Yaskawa INFORM job: BATMAN_NEW2.JBI

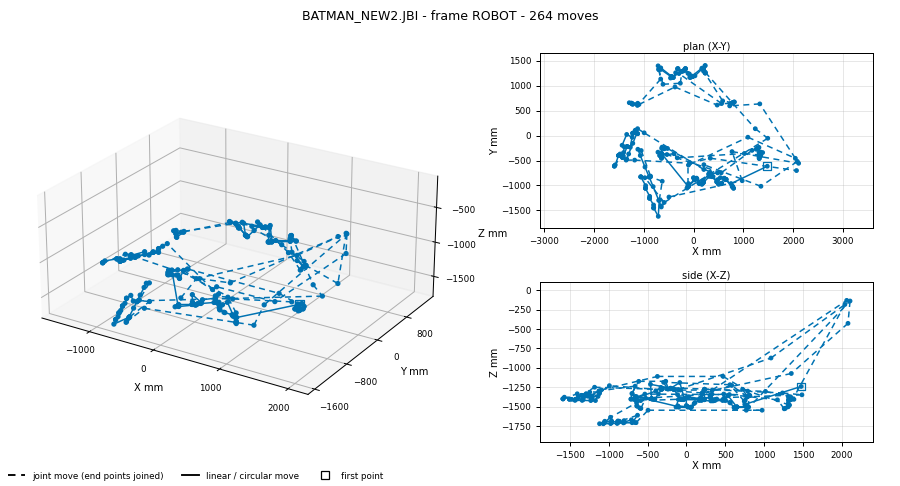
[picture p0: tool path of BATMAN_NEW2.JBI in frame ROBOT, 264 of 264 moves have a stored position in this frame; points joined in program order, loops and branches not executed]
/JOB
//NAME BATMAN_NEW2
///FOLDERNAME KRIS-SCIANA
//POS
///NPOS 316,316,264,16,0,0
///TOOL 0
///POSTYPE ROBOT
///RECTAN
///RCONF 0,0,0,0,0,0,0,0,0,0,0,0,0,0,0,0,0,0,0,0,0,0,0,0
C00000=1479.209,-614.254,-1239.827,11.6326,33.9671,-178.8219
C00001=751.878,-962.551,-1470.637,-9.9278,21.9341,47.3593
C00002=782.343,-1021.883,-1501.453,-6.5198,31.4589,38.6711
C00003=782.349,-1021.901,-1508.593,-6.5211,31.4595,38.6707
C00004=782.343,-1021.883,-1501.453,-6.5198,31.4589,38.6711
C00005=772.436,-1031.632,-1503.007,-6.5210,31.4603,38.6751
C00006=782.343,-1021.883,-1501.453,-6.5198,31.4589,38.6711
C00007=651.465,-878.509,-1502.529,-6.5193,31.4567,38.6726
C00008=649.681,-879.962,-1505.034,-6.5204,31.4570,38.6688
C00009=649.679,-879.971,-1512.967,-6.5216,31.4579,38.6721
C00010=649.681,-879.962,-1505.034,-6.5204,31.4570,38.6688
C00011=638.496,-885.487,-1507.904,-6.5213,31.4572,38.6690
C00012=649.681,-879.962,-1505.034,-6.5204,31.4570,38.6688
C00013=536.093,-844.110,-1358.224,-6.5194,31.4565,38.6698
C00014=485.208,-882.506,-1390.226,-6.5180,31.4566,38.6722
C00015=469.831,-925.588,-1412.310,-6.5196,31.4595,38.6720
C00016=469.838,-925.615,-1422.209,-6.5208,31.4607,38.6737
C00017=469.831,-925.588,-1412.310,-6.5196,31.4595,38.6720
C00018=460.916,-939.180,-1415.903,-6.5217,31.4610,38.6723
C00019=469.831,-925.588,-1412.310,-6.5196,31.4595,38.6720
C00020=390.944,-821.413,-1401.907,-6.5189,31.4593,38.6711
C00021=370.304,-823.702,-1415.949,-6.5184,31.4594,38.6679
C00022=370.309,-823.695,-1427.366,-6.5174,31.4589,38.6696
C00023=370.304,-823.702,-1415.949,-6.5184,31.4594,38.6679
C00024=362.481,-832.843,-1419.419,-6.5181,31.4591,38.6684
C00025=370.304,-823.702,-1415.949,-6.5184,31.4594,38.6679
C00026=304.377,-775.536,-1384.314,-6.5183,31.4594,38.6652
C00027=190.919,-901.974,-1384.308,6.6118,30.8401,128.8238
C00028=195.878,-934.762,-1411.685,6.6092,30.8405,128.8212
C00029=195.887,-934.767,-1420.325,6.6101,30.8407,128.8263
C00030=195.878,-934.762,-1411.685,6.6092,30.8405,128.8212
C00031=202.495,-948.084,-1414.851,6.6099,30.8403,128.8223
C00032=195.878,-934.762,-1411.685,6.6092,30.8405,128.8212
C00033=-1.386,-846.899,-1381.133,6.6069,30.8405,134.1399
C00034=-1.384,-846.902,-1485.292,6.6071,30.8406,134.1408
C00035=18.120,-884.199,-1503.049,6.6086,30.8410,134.1399
C00036=18.115,-884.194,-1511.506,6.6087,30.8409,134.1387
C00037=18.120,-884.199,-1503.049,6.6086,30.8410,134.1399
C00038=26.172,-895.008,-1505.663,6.6092,30.8415,134.1385
C00039=18.120,-884.199,-1503.049,6.6086,30.8410,134.1399
C00040=-111.813,-1001.782,-1489.786,6.6089,30.8396,134.1409
C00041=-110.516,-1020.985,-1499.218,6.6089,30.8402,134.1417
C00042=-110.523,-1020.998,-1507.131,6.6095,30.8409,134.1397
C00043=-110.516,-1020.985,-1499.218,6.6089,30.8402,134.1417
C00044=-104.498,-1031.543,-1502.310,6.6099,30.8394,134.1431
C00045=-110.516,-1020.985,-1499.218,6.6089,30.8402,134.1417
C00046=-641.458,-364.123,-1372.142,-0.2839,36.0778,31.9819
C00047=-662.744,-397.701,-1394.268,-0.2832,36.0779,31.9810
C00048=-662.752,-397.694,-1404.858,-0.2824,36.0779,31.9809
C00049=-662.744,-397.701,-1394.268,-0.2832,36.0779,31.9810
C00050=-686.425,-397.683,-1394.265,-0.2810,36.0766,31.9839
C00051=-662.744,-397.701,-1394.268,-0.2832,36.0779,31.9810
C00052=-395.220,-362.676,-1299.812,-0.2837,36.0781,31.9812
C00053=-328.978,-445.538,-1251.827,-0.2820,36.0777,31.9846
C00054=1019.066,-358.271,-1303.588,-0.7093,36.3388,173.5111
C00055=1312.502,-388.638,-1368.088,-0.7090,36.3391,143.8761
C00056=1330.261,-409.263,-1395.611,-0.7097,36.3382,143.8752
C00057=1330.266,-409.258,-1408.665,-0.7105,36.3381,143.8742
C00058=1330.261,-409.263,-1395.611,-0.7097,36.3382,143.8752
C00059=1359.166,-409.282,-1395.624,-0.7081,36.3381,143.8755
C00060=1330.261,-409.263,-1395.611,-0.7097,36.3382,143.8752
C00061=1346.256,-330.236,-1377.208,-0.7085,36.3387,143.8760
C00062=1385.768,-339.505,-1405.683,-0.7074,36.3385,143.8819
C00063=1349.259,-407.967,-1405.698,-0.7099,36.3376,143.8723
C00064=1344.221,-409.875,-1407.374,-0.7109,36.3390,143.8722
C00065=1319.007,-459.412,-1408.358,-0.7127,36.3385,143.8707
C00066=1316.585,-457.113,-1411.355,-0.7151,36.3388,143.8640
C00067=1314.211,-431.828,-1419.878,-0.7170,36.3383,163.2059
C00068=1313.610,-343.846,-1457.563,-0.7163,36.3370,163.2057
C00069=1312.103,-236.565,-1499.789,-0.7202,36.3387,-169.8421
C00070=1305.396,-239.618,-1503.423,-0.7150,36.3420,-169.8387
C00071=1273.863,-258.154,-1521.213,-0.7182,36.3419,-169.8425
C00072=1267.468,-262.937,-1524.998,1.6686,33.5135,174.0856
C00073=1260.689,-274.030,-1527.843,2.4139,32.4267,168.8905
C00074=1172.939,-295.478,-1411.838,2.4149,32.4260,168.8924
C00075=553.926,-745.251,-1344.470,9.9580,22.3671,144.0884
C00076=-536.407,-379.228,-1337.930,-3.7346,30.6001,32.3556
C00077=-716.129,-331.806,-1403.803,-3.7368,30.5972,32.3471
C00078=-681.265,-398.771,-1403.765,-3.7327,30.5994,32.3525
C00079=-676.698,-399.723,-1405.572,-3.7330,30.6001,32.3555
C00080=-644.842,-456.418,-1406.142,-3.7344,30.5987,32.3598
C00081=-644.657,-446.831,-1409.438,-3.7314,30.5969,32.3583
C00082=-644.722,-424.014,-1417.852,6.8176,41.7160,38.5658
C00083=-643.136,-351.092,-1448.860,6.8129,41.7188,38.5566
C00084=-641.376,-256.892,-1488.844,6.7765,41.4627,22.9424
C00085=-633.859,-231.097,-1495.754,6.8200,41.7180,-9.8008
C00086=-601.904,-250.806,-1517.185,12.2909,40.7284,-6.2420
C00087=-592.469,-255.965,-1521.502,6.8207,41.7173,-9.7972
C00088=-587.357,-263.536,-1522.796,6.8200,41.7194,22.2662
C00089=-524.640,-257.672,-1391.051,6.8232,41.7195,-9.7941
C00090=328.849,-733.445,-1337.611,2.7644,30.8890,70.6747
C00091=338.434,-795.853,-1424.595,2.7651,30.8864,70.6725
C00092=347.583,-803.582,-1424.840,2.7653,30.8871,70.6737
C00093=465.379,-931.076,-1420.407,2.7642,30.8893,70.6731
C00094=500.376,-972.906,-1419.509,2.7673,30.8880,70.6771
C00095=502.727,-974.471,-1420.148,2.7642,30.8895,70.6782
C00096=558.221,-962.583,-1445.651,29.9139,35.7052,85.7904
C00097=565.911,-953.297,-1452.392,19.5066,42.2165,79.2495
C00098=613.155,-854.018,-1511.422,19.5140,42.2128,79.2557
C00099=619.427,-858.037,-1512.184,3.7149,38.7712,68.9600
C00100=645.632,-884.392,-1510.752,-0.5869,30.5405,66.8336
C00101=773.676,-1024.707,-1508.152,1.6006,33.1200,67.9710
C00102=802.105,-1054.466,-1506.146,3.6687,32.7293,69.0093
C00103=802.122,-1056.982,-1354.174,6.2530,30.6739,70.3394
C00104=481.154,-746.898,-1337.541,6.2536,30.6743,70.3404
C00105=303.930,-769.190,-1354.154,12.5353,29.0330,117.3688
C00106=330.080,-800.270,-1423.712,12.5361,29.0314,117.3697
C00107=314.779,-818.672,-1426.191,12.5335,29.0333,117.3718
C00108=194.426,-946.689,-1419.614,12.5356,29.0342,117.3720
C00109=168.116,-974.806,-1418.609,12.5340,29.0299,117.3778
C00110=164.045,-973.945,-1418.599,12.5354,29.0311,117.3765
C00111=111.592,-964.862,-1447.278,-20.8945,38.2915,98.4113
C00112=98.760,-940.057,-1460.333,-8.8483,43.5864,106.1648
C00113=66.281,-867.817,-1502.677,-8.8480,43.5869,106.1636
C00114=58.359,-853.021,-1511.906,-8.8470,43.5851,106.1701
C00115=48.723,-860.440,-1512.145,-8.7706,29.7610,106.6794
C00116=-100.605,-1019.492,-1507.714,-8.7679,29.7616,106.6753
C00117=-133.982,-1054.517,-1505.581,-8.7689,29.7575,106.6753
C00118=-104.193,-961.904,-1408.358,-8.7704,29.7603,106.6778
C00119=-104.195,-589.697,-1279.272,-8.7711,29.7586,106.6768
C00120=1089.919,-31.439,-873.125,-36.7541,69.9873,137.0084
///RCONF 0,0,0,0,1,0,0,0,0,0,0,0,0,0,0,0,0,0,0,0,0,0,0,0
C00121=2042.728,-454.958,-183.433,1.6788,-19.8065,-6.7510
C00122=1329.047,637.602,-1479.857,8.0540,25.5528,30.8439
///RCONF 0,0,0,0,0,0,0,0,0,0,0,0,0,0,0,0,0,0,0,0,0,0,0,0
C00123=724.107,597.545,-1276.344,-3.2635,41.6684,-140.4024
C00124=785.383,659.459,-1372.820,-3.2632,41.6678,-140.4000
C00125=792.753,652.576,-1383.361,-3.2644,41.6697,-140.4060
C00126=785.383,659.459,-1372.820,-3.2632,41.6678,-140.4000
C00127=780.124,673.327,-1385.992,-3.2593,41.6675,-140.3923
C00128=785.383,659.459,-1372.820,-3.2632,41.6678,-140.4000
C00129=583.065,697.790,-1226.639,-3.1675,40.5415,-139.9875
C00130=200.134,1294.158,-1339.988,10.2608,31.0598,-45.0576
C00131=172.748,1341.866,-1398.059,10.2620,31.0622,-45.0581
C00132=172.750,1341.856,-1411.003,10.2608,31.0619,-45.0612
C00133=172.748,1341.866,-1398.059,10.2620,31.0622,-45.0581
C00134=162.053,1360.361,-1403.672,10.2607,31.0636,-45.0654
C00135=172.748,1341.866,-1398.059,10.2620,31.0622,-45.0581
C00136=26.821,1201.359,-1372.636,10.2610,31.0614,-45.0581
C00137=-26.114,1184.722,-1395.825,10.2614,31.0609,-45.0571
C00138=-26.119,1184.747,-1409.910,10.2622,31.0622,-45.0567
C00139=-26.114,1184.722,-1395.825,10.2614,31.0609,-45.0571
C00140=-38.557,1201.364,-1401.881,10.2611,31.0613,-45.0602
C00141=-26.114,1184.722,-1395.825,10.2614,31.0609,-45.0571
C00142=-85.944,1239.452,-1189.279,10.2632,31.0602,-45.0547
C00143=-202.376,1302.359,-1263.326,10.2654,31.0601,-39.0783
C00144=-202.377,1302.375,-1273.759,10.2665,31.0600,-39.0755
C00145=-202.376,1302.359,-1263.326,10.2654,31.0601,-39.0783
C00146=-213.401,1315.412,-1266.159,10.2653,31.0594,-39.0754
C00147=-202.376,1302.359,-1263.326,10.2654,31.0601,-39.0783
C00148=-463.805,1156.888,-1211.984,5.4408,32.3182,-121.2144
C00149=-448.455,1180.872,-1396.312,5.4420,32.3182,-121.2130
C00150=-448.461,1180.875,-1405.887,5.4414,32.3181,-121.2136
C00151=-448.455,1180.872,-1396.312,5.4420,32.3182,-121.2130
C00152=-438.739,1194.365,-1399.533,5.4424,32.3182,-121.2152
C00153=-448.455,1180.872,-1396.312,5.4420,32.3182,-121.2130
C00154=-657.730,1329.361,-1367.973,5.4433,32.3188,-121.2093
C00155=-663.299,1347.249,-1396.310,5.4469,32.3207,-121.2088
C00156=-663.288,1347.263,-1404.262,5.4479,32.3220,-121.2052
C00157=-663.299,1347.249,-1396.310,5.4469,32.3207,-121.2088
C00158=-654.469,1361.022,-1397.928,5.4472,32.3207,-121.2069
C00159=-663.299,1347.249,-1396.310,5.4469,32.3207,-121.2088
C00160=-698.479,1323.579,-1333.586,5.4477,32.3218,-121.2085
C00161=-661.200,1136.351,-1235.695,5.4453,32.3209,-21.5885
C00162=-1128.608,606.997,-1296.811,5.4402,32.3220,-21.6018
C00163=-1245.560,650.345,-1363.191,5.4391,32.3216,-21.6043
C00164=-1253.840,659.612,-1369.532,5.4396,32.3086,-21.6048
C00165=-1245.560,650.345,-1363.191,5.4391,32.3216,-21.6043
C00166=-1255.518,641.298,-1375.299,5.4388,32.3217,-21.6053
C00167=-1245.560,650.345,-1363.191,5.4391,32.3216,-21.6043
C00168=-1122.499,650.360,-1312.804,5.4384,32.3212,-21.6061
C00169=-1246.019,650.333,-1312.805,-5.9814,50.4641,-44.8970
C00170=-1292.168,661.169,-1333.261,-5.9804,50.4648,-44.8927
C00171=-1228.022,632.044,-1400.190,-5.9775,50.4666,-44.8867
C00172=-1221.375,630.664,-1404.684,9.2048,37.0985,-34.2692
C00173=-1097.819,626.024,-1284.700,9.2046,37.0985,-34.2704
C00174=-374.253,977.072,-1110.582,-16.3615,18.9747,-168.4330
C00175=472.792,614.034,-1110.590,-6.3310,51.0848,-162.4334
C00176=790.077,666.826,-1299.714,-6.3326,51.0845,-162.4374
C00177=816.173,675.910,-1358.543,-6.3341,51.0842,-155.2649
C00178=816.189,675.286,-1355.228,-6.3386,51.0862,-155.2697
C00179=757.591,647.487,-1417.938,-6.3356,51.0871,-155.2637
C00180=745.147,646.476,-1430.103,-12.0666,41.5969,-159.4258
C00181=561.133,644.284,-1217.351,-12.0669,41.5966,-159.4267
C00182=-294.154,1247.220,-1186.692,-14.7086,35.8481,-158.3060
C00183=-242.562,1288.482,-1273.150,-14.2330,35.5827,-141.3920
C00184=-312.355,1343.168,-1271.625,-14.2215,35.5974,-141.3854
C00185=-318.403,1347.498,-1273.796,-14.2220,35.5979,-141.3873
C00186=-322.722,1341.692,-1279.720,-14.2224,35.5978,-157.9766
C00187=-360.894,1263.349,-1337.011,-14.2220,35.5972,-157.9819
C00188=-406.929,1169.712,-1402.159,-14.2205,35.5995,-157.9818
C00189=-409.686,1166.190,-1406.287,-14.2225,35.5992,-147.9816
C00190=-417.767,1173.056,-1406.551,-14.2208,35.5994,-147.9812
C00191=-440.474,1190.413,-1406.120,-14.2202,35.6028,-144.4913
C00192=-660.245,1361.072,-1403.707,-14.2205,35.6058,-144.4916
C00193=-713.508,1401.790,-1402.114,-14.2216,35.6049,-144.4985
C00194=-702.785,1334.590,-1330.560,-14.2225,35.6052,-144.4992
C00195=-615.113,1031.882,-1174.072,-14.2237,35.6047,-144.5023
C00196=-266.790,1052.428,-1172.785,14.1594,35.6599,-52.4229
C00197=-234.621,1290.298,-1271.352,14.1573,35.6533,-52.4193
C00198=-170.266,1343.198,-1274.471,14.1621,35.6578,-52.4205
C00199=-163.350,1347.913,-1274.487,14.1614,35.6572,-52.4200
C00200=-161.403,1342.862,-1281.279,7.3802,43.3671,-41.1599
C00201=-113.870,1250.739,-1345.243,7.3795,43.3689,-41.1646
C00202=-75.578,1173.045,-1403.534,7.3827,43.3703,-41.1594
C00203=-71.378,1165.451,-1408.302,7.3856,43.3696,-41.1548
C00204=-59.197,1175.793,-1409.651,4.6384,38.1537,-42.8411
C00205=-35.448,1195.776,-1410.312,4.6465,38.1543,-47.5801
C00206=166.563,1354.922,-1410.948,4.6441,38.1493,-47.5848
C00207=227.339,1402.932,-1410.926,4.6442,38.1483,-47.5854
C00208=233.128,1408.173,-1410.916,4.6445,38.1490,-47.5846
C00209=233.146,1258.590,-1276.348,4.6463,38.1495,-47.5846
C00210=233.273,1258.338,-1276.378,4.6470,38.1496,-47.5838
C00211=233.273,1258.338,-1276.378,4.6470,38.1496,-47.5838
C00212=233.248,1273.531,-1276.386,4.6460,38.1499,-47.5825
C00213=1238.436,139.129,-1323.509,-1.5927,36.9682,-135.2428
C00214=1488.778,-52.476,-1347.695,27.2487,24.5669,-70.7938
C00215=-591.325,-1341.846,-1422.510,-0.6043,40.8297,16.7434
C00216=-978.344,-845.186,-1637.203,-0.6000,40.8277,16.7477
C00217=-1060.712,-827.560,-1707.784,-0.5964,40.8264,16.7530
C00218=-1060.716,-827.565,-1719.613,-0.5979,40.8266,16.7496
C00219=-1060.712,-827.560,-1707.784,-0.5964,40.8264,16.7530
C00220=-1076.749,-827.566,-1707.781,-0.5968,40.8274,16.7526
C00221=-1060.712,-827.560,-1707.784,-0.5964,40.8264,16.7530
C00222=-964.064,-1003.361,-1685.365,-0.5978,40.8280,16.7499
C00223=-967.258,-1055.832,-1705.053,-0.5976,40.8279,16.7488
C00224=-967.265,-1055.827,-1717.171,-0.5974,40.8281,16.7474
C00225=-967.258,-1055.832,-1705.053,-0.5976,40.8279,16.7488
C00226=-984.967,-1055.847,-1705.045,-0.5977,40.8287,16.7479
C00227=-967.258,-1055.832,-1705.053,-0.5976,40.8279,16.7488
C00228=-883.106,-1217.890,-1684.422,-0.5980,40.8275,16.7460
C00229=-884.555,-1256.605,-1703.312,-0.5986,40.8276,16.7466
C00230=-884.543,-1256.571,-1713.321,-0.5947,40.8260,16.7508
C00231=-884.555,-1256.605,-1703.312,-0.5986,40.8276,16.7466
C00232=-901.563,-1256.594,-1703.316,-0.6002,40.8264,16.7423
C00233=-884.555,-1256.605,-1703.312,-0.5986,40.8276,16.7466
C00234=-804.394,-1392.262,-1680.447,-0.5972,40.8269,16.7457
C00235=-802.318,-1451.144,-1699.808,-0.5973,40.8272,16.7464
C00236=-802.295,-1451.144,-1709.722,-0.5981,40.8252,16.7458
C00237=-802.318,-1451.144,-1699.808,-0.5973,40.8272,16.7464
C00238=-820.040,-1451.129,-1699.830,-0.5958,40.8269,16.7480
C00239=-802.318,-1451.144,-1699.808,-0.5973,40.8272,16.7464
C00240=-709.611,-1620.676,-1670.338,-0.5978,40.8273,16.7476
C00241=-689.604,-1294.748,-1695.996,-0.5975,40.8268,16.7459
C00242=-689.614,-1294.765,-1707.440,-0.5999,40.8277,16.7418
C00243=-689.604,-1294.748,-1695.996,-0.5975,40.8268,16.7459
C00244=-710.807,-1294.753,-1696.008,-0.5986,40.8259,16.7454
C00245=-689.604,-1294.748,-1695.996,-0.5975,40.8268,16.7459
C00246=-630.511,-916.030,-1610.753,-0.6017,40.8266,16.7401
C00247=-868.430,-829.435,-1692.124,-0.6028,40.8258,16.7353
C00248=-892.870,-831.979,-1714.985,-0.5981,40.8255,16.7444
C00249=-976.713,-630.080,-1718.549,-0.6011,40.8246,16.7412
C00250=-1071.217,-398.415,-1720.690,-0.6000,40.8208,16.7397
C00251=-1119.996,-273.264,-1720.027,-0.6007,40.8208,16.7405
C00252=-1052.650,-299.020,-1688.341,-0.6009,40.8211,16.7408
C00253=-865.284,-812.787,-1688.334,-0.6039,40.8202,42.9608
C00254=-892.749,-830.002,-1713.253,-0.5986,40.8166,42.9666
C00255=-812.172,-1024.012,-1709.563,-0.6014,40.8165,42.9567
C00256=-700.538,-1299.832,-1707.155,-0.6008,40.8192,42.9610
C00257=-657.041,-1411.182,-1706.542,-0.5992,40.8178,42.9644
C00258=-649.131,-1432.542,-1706.544,-0.5977,40.8180,42.9663
C00259=-495.179,-1232.483,-1546.245,-0.5800,40.8231,42.9777
C00260=975.318,-905.329,-1546.300,2.7447,40.6858,121.3068
C00261=771.357,-320.253,-1546.238,-0.5794,40.8236,124.0583
///RCONF 0,0,0,0,1,0,0,0,0,0,0,0,0,0,0,0,0,0,0,0,0,0,0,0
C00262=2108.910,-555.323,-138.194,2.1712,-19.6918,-3.5371
///RCONF 0,0,0,0,0,0,0,0,0,0,0,0,0,0,0,0,0,0,0,0,0,0,0,0
C00263=2082.559,-517.688,-426.187,17.7899,-11.9984,-30.1124
C00264=1351.715,-1016.627,-1072.730,14.7650,1.4143,-53.7135
C00265=205.703,-583.482,-1322.085,9.2825,24.4184,-95.9833
C00266=203.961,-679.195,-1324.426,-9.5613,21.9567,95.9050
C00267=-993.168,56.729,-1229.540,-0.2104,49.9239,-21.9207
C00268=-1124.976,139.813,-1330.335,5.3125,39.0598,-25.3648
C00269=-1217.958,48.598,-1401.440,5.3913,38.9364,-25.3168
C00270=-1222.465,48.743,-1409.263,5.3874,38.9378,-25.3223
C00271=-1222.459,48.730,-1420.612,5.3858,38.9371,-25.3242
C00272=-1222.465,48.743,-1409.263,5.3874,38.9378,-25.3223
C00273=-1239.080,48.748,-1409.236,5.3856,38.9399,-25.3266
C00274=-1222.465,48.743,-1409.263,5.3874,38.9378,-25.3223
C00275=-1271.414,-233.653,-1365.903,5.3880,38.9368,-25.3214
C00276=-1335.102,-218.968,-1407.739,5.3747,38.9270,-25.3244
C00277=-1335.110,-218.964,-1419.095,5.3738,38.9278,-25.3274
C00278=-1335.102,-218.968,-1407.739,5.3747,38.9270,-25.3244
C00279=-1351.938,-218.955,-1407.734,5.3749,38.9273,-25.3233
C00280=-1335.102,-218.968,-1407.739,5.3747,38.9270,-25.3244
C00281=-1410.796,-411.626,-1397.644,5.3751,38.9281,-25.3225
C00282=-1428.227,-437.232,-1406.270,5.3763,38.9287,-25.3214
C00283=-1428.230,-437.231,-1419.122,5.3758,38.9290,-25.3227
C00284=-1428.227,-437.232,-1406.270,5.3763,38.9287,-25.3214
C00285=-1445.183,-437.215,-1406.274,5.3770,38.9284,-25.3233
C00286=-1428.227,-437.232,-1406.270,5.3763,38.9287,-25.3214
C00287=-1478.764,-369.056,-1406.265,5.3746,38.9285,-25.3278
C00288=-1508.274,-399.507,-1403.549,5.3752,38.9282,-25.3298
C00289=-1508.284,-399.505,-1415.860,5.3764,38.9286,-25.3265
C00290=-1508.274,-399.507,-1403.549,5.3752,38.9282,-25.3298
C00291=-1525.499,-399.503,-1403.534,5.3741,38.9288,-25.3312
C00292=-1508.274,-399.507,-1403.549,5.3752,38.9282,-25.3298
C00293=-1573.700,-586.702,-1378.129,5.3749,38.9274,-25.3303
C00294=-1591.625,-610.872,-1399.727,5.3751,38.9284,-25.3300
C00295=-1591.607,-610.857,-1410.848,5.3774,38.9278,-25.3276
C00296=-1591.625,-610.872,-1399.727,5.3751,38.9284,-25.3300
C00297=-1607.585,-610.886,-1399.726,5.3748,38.9284,-25.3293
C00298=-1591.625,-610.872,-1399.727,5.3751,38.9284,-25.3300
C00299=-1407.614,-340.295,-1334.283,5.3763,38.9277,-25.3283
C00300=-1393.545,-225.421,-1380.034,5.3755,38.9268,-25.3271
C00301=-1436.319,-192.923,-1419.519,-0.6441,37.4048,-43.4681
C00302=-1343.970,24.204,-1419.685,-0.6458,37.4045,-43.4729
C00303=-1233.172,-33.364,-1421.676,-0.6450,37.4042,-43.4706
C00304=-1172.683,108.529,-1421.468,-0.6415,37.4057,-43.4715
C00305=-1123.867,39.567,-1327.748,-0.6454,37.4059,-43.4725
C00306=-1123.867,39.567,-1327.748,-0.6454,37.4059,-43.4725
C00307=-1139.614,46.545,-1367.957,-0.6485,37.4091,-15.9314
C00308=-1221.149,-154.590,-1364.989,-0.6505,37.4071,-15.9367
C00309=-1304.293,-367.690,-1359.056,-0.6521,37.4085,-15.9430
C00310=-1343.286,-469.596,-1355.805,-0.6535,37.4062,-15.9492
C00311=-1354.672,-491.189,-1354.002,-0.6534,37.4048,-15.9508
C00312=-1184.082,-491.180,-1249.860,-0.6521,37.4040,-15.9519
C00313=-78.969,-554.378,-1286.716,1.4249,23.3229,2.1506
C00314=333.912,-453.248,-1285.762,1.2790,23.3311,46.5433
C00315=2065.993,-701.065,-130.284,1.6748,-19.7957,-6.8086
BC00000=506.026,2197.799,889.024
BC00001=1028.973,2071.524,879.905
BC00002=1028.973,2071.524,879.905
BC00003=1028.973,2071.524,879.905
BC00004=1028.973,2071.524,879.905
BC00005=1028.973,2071.524,879.905
BC00006=1028.973,2071.524,879.905
BC00007=1028.973,2071.524,879.905
BC00008=1028.973,2071.524,879.905
BC00009=1028.973,2071.524,879.905
BC00010=1028.973,2071.524,879.905
BC00011=1028.973,2071.524,879.905
BC00012=1028.973,2071.524,879.905
BC00013=1028.973,2071.524,879.905
BC00014=1028.973,2071.524,879.905
BC00015=1028.973,2071.524,879.905
BC00016=1028.973,2071.524,879.905
BC00017=1028.973,2071.524,879.905
BC00018=1028.973,2071.524,879.905
BC00019=1028.973,2071.524,879.905
BC00020=1028.973,2071.524,879.905
BC00021=1028.973,2071.524,879.905
BC00022=1028.973,2071.524,879.905
BC00023=1028.973,2071.524,879.905
BC00024=1028.973,2071.524,879.905
BC00025=1028.973,2071.524,879.905
BC00026=1028.973,2071.524,879.905
BC00027=1028.973,2071.524,879.905
BC00028=1028.973,2071.524,879.905
BC00029=1028.973,2071.524,879.905
BC00030=1028.973,2071.524,879.905
BC00031=1028.973,2071.524,879.905
BC00032=1028.973,2071.524,879.905
BC00033=1028.973,2071.524,879.905
BC00034=1028.973,2071.524,879.905
BC00035=1028.973,2071.524,879.905
BC00036=1028.973,2071.524,879.905
BC00037=1028.973,2071.524,879.905
BC00038=1028.973,2071.524,879.905
BC00039=1028.973,2071.524,879.905
BC00040=1028.973,2071.524,879.905
BC00041=1028.973,2071.524,879.905
BC00042=1028.973,2071.524,879.905
BC00043=1028.973,2071.524,879.905
BC00044=1028.973,2071.524,879.905
BC00045=1028.973,2071.524,879.905
BC00046=1028.973,2071.524,879.905
BC00047=1028.973,2071.524,879.905
BC00048=1028.973,2071.524,879.905
BC00049=1028.973,2071.524,879.905
BC00050=1028.973,2071.524,879.905
BC00051=1028.973,2071.524,879.905
BC00052=1028.973,2071.524,879.905
BC00053=1028.973,2071.524,879.905
BC00054=1028.973,2071.524,879.905
BC00055=1028.973,2071.524,879.905
BC00056=1028.973,2071.524,879.905
BC00057=1028.973,2071.524,879.905
BC00058=1028.973,2071.524,879.905
BC00059=1028.973,2071.524,879.905
BC00060=1028.973,2071.524,879.905
BC00061=1028.973,2071.524,879.905
BC00062=1028.973,2071.524,879.905
BC00063=1028.973,2071.524,879.905
BC00064=1028.973,2071.524,879.905
BC00065=1028.973,2071.524,879.905
BC00066=1028.973,2071.524,879.905
BC00067=1028.973,2071.524,879.905
BC00068=1028.973,2071.524,879.905
BC00069=1028.973,2071.524,879.905
BC00070=1028.973,2071.524,879.905
BC00071=1028.973,2071.524,879.905
BC00072=1028.979,2071.524,879.911
BC00073=1028.979,2071.524,879.911
BC00074=1028.979,2071.524,879.911
BC00075=1028.979,2071.531,1132.335
BC00076=1028.979,2071.531,879.905
BC00077=1028.979,2071.531,879.905
BC00078=1028.979,2071.531,879.905
BC00079=1028.979,2071.531,879.905
BC00080=1028.979,2071.531,879.905
BC00081=1028.979,2071.531,879.905
BC00082=1028.979,2071.531,879.905
BC00083=1028.979,2071.531,879.905
BC00084=1028.979,2071.531,879.905
BC00085=1028.979,2071.531,879.905
BC00086=1028.979,2071.531,879.905
BC00087=1028.979,2071.531,879.905
BC00088=1028.979,2071.531,879.905
BC00089=1028.979,2071.531,879.905
BC00090=1028.979,2071.531,879.905
BC00091=1028.979,2071.531,879.905
BC00092=1028.979,2071.531,879.905
BC00093=1028.979,2071.531,879.905
BC00094=1028.979,2071.531,879.905
BC00095=1028.979,2071.531,879.905
BC00096=1028.979,2071.531,879.905
BC00097=1028.979,2071.531,879.905
BC00098=1028.979,2071.531,879.905
BC00099=1028.979,2071.531,879.905
BC00100=1028.973,2071.537,879.898
BC00101=1028.979,2071.531,879.905
BC00102=1028.979,2071.531,879.905
BC00103=1028.979,2071.531,879.905
BC00104=1028.979,2071.531,879.905
BC00105=1028.979,2071.531,879.905
BC00106=1028.979,2071.531,879.905
BC00107=1028.979,2071.531,879.905
BC00108=1028.979,2071.531,879.905
BC00109=1028.979,2071.531,879.905
BC00110=1028.979,2071.531,879.905
BC00111=1028.979,2071.531,879.905
BC00112=1028.979,2071.531,879.905
BC00113=1028.979,2071.531,879.905
BC00114=1028.979,2071.531,879.905
BC00115=1028.979,2071.531,879.905
BC00116=1028.979,2071.531,879.905
BC00117=1028.979,2071.531,879.905
BC00118=1028.979,2071.531,879.905
BC00119=1028.979,2071.531,1313.400
BC00120=705.175,35.017,1952.866
BC00121=786.422,38.780,1999.645
BC00122=786.422,38.780,1999.645
BC00123=1602.623,32.856,1148.414
BC00124=1602.623,32.856,1148.414
BC00125=1602.623,32.856,1148.414
BC00126=1602.623,32.856,1148.414
BC00127=1602.623,32.856,1148.414
BC00128=1602.623,32.856,1148.414
BC00129=1602.623,32.856,1148.414
BC00130=1602.623,32.856,1148.414
BC00131=1602.623,32.856,1148.414
BC00132=1602.623,32.856,1148.414
BC00133=1602.623,32.856,1148.414
BC00134=1602.623,32.856,1148.414
BC00135=1602.623,32.856,1148.414
BC00136=1602.623,32.856,1148.414
BC00137=1602.623,32.856,1148.414
BC00138=1602.623,32.856,1148.414
BC00139=1602.623,32.856,1148.414
BC00140=1602.623,32.856,1148.414
BC00141=1602.623,32.856,1148.414
BC00142=1602.623,32.856,1148.414
BC00143=1602.623,32.856,1148.414
BC00144=1602.623,32.856,1148.414
BC00145=1602.623,32.856,1148.414
BC00146=1602.623,32.856,1148.414
BC00147=1602.623,32.856,1148.414
BC00148=1602.623,32.856,1148.414
BC00149=1602.623,32.856,1148.414
BC00150=1602.623,32.856,1148.414
BC00151=1602.623,32.856,1148.414
BC00152=1602.623,32.856,1148.414
BC00153=1602.623,32.856,1148.414
BC00154=1602.623,32.856,1148.414
BC00155=1602.623,32.856,1148.414
BC00156=1602.623,32.856,1148.414
BC00157=1602.623,32.856,1148.414
BC00158=1602.623,32.856,1148.414
BC00159=1602.623,32.856,1148.414
BC00160=1602.623,32.856,1148.414
BC00161=1602.623,32.856,1148.414
BC00162=1602.623,32.856,1148.414
BC00163=1602.623,32.856,1148.414
BC00164=1602.617,32.863,1148.408
BC00165=1602.623,32.856,1148.414
BC00166=1602.623,32.856,1148.414
BC00167=1602.623,32.856,1148.414
BC00168=1602.623,32.856,1148.414
BC00169=1602.623,32.856,1148.414
BC00170=1602.623,32.856,1148.414
BC00171=1602.623,32.856,1148.414
BC00172=1602.623,32.856,1148.414
BC00173=1602.623,32.856,1148.414
BC00174=1602.617,32.856,1148.408
BC00175=1602.617,32.856,1148.408
BC00176=1602.617,32.856,1148.408
BC00177=1602.617,32.856,1148.408
BC00178=1602.610,32.863,1148.395
BC00179=1602.610,32.863,1148.395
BC00180=1602.610,32.863,1148.395
BC00181=1602.610,32.863,1148.395
BC00182=1602.610,32.863,1148.395
BC00183=1602.610,32.863,1148.395
BC00184=1602.610,32.863,1148.391
BC00185=1602.610,32.863,1148.391
BC00186=1602.610,32.863,1148.391
BC00187=1602.610,32.863,1148.391
BC00188=1602.610,32.863,1148.391
BC00189=1602.610,32.863,1148.391
BC00190=1602.610,32.863,1148.391
BC00191=1602.610,32.863,1148.391
BC00192=1602.610,32.863,1148.391
BC00193=1602.610,32.863,1148.391
BC00194=1602.610,32.863,1148.391
BC00195=1602.610,32.863,1148.391
BC00196=1602.610,32.863,1148.391
BC00197=1602.617,32.863,1148.387
BC00198=1602.617,32.863,1148.387
BC00199=1602.617,32.863,1148.387
BC00200=1602.617,32.863,1148.387
BC00201=1602.617,32.863,1148.387
BC00202=1602.617,32.863,1148.387
BC00203=1602.617,32.863,1148.387
BC00204=1602.617,32.863,1148.387
BC00205=1602.617,32.863,1148.387
BC00206=1602.617,32.863,1148.387
BC00207=1602.617,32.863,1148.387
BC00208=1602.617,32.863,1148.387
BC00209=1602.617,32.863,1148.387
BC00210=1602.617,32.863,1960.335
BC00211=2287.550,32.863,1960.335
BC00212=2172.832,3214.278,1960.335
BC00213=752.940,3214.278,1960.335
BC00214=766.746,3215.828,1976.542
BC00215=1984.483,3218.041,658.883
BC00216=1984.483,2448.792,658.883
BC00217=1984.483,2448.792,658.883
BC00218=1984.483,2448.792,658.883
BC00219=1984.483,2448.792,658.883
BC00220=1984.483,2448.792,658.883
BC00221=1984.483,2448.792,658.883
BC00222=1984.483,2448.792,658.883
BC00223=1984.483,2448.792,658.883
BC00224=1984.483,2448.792,658.883
BC00225=1984.483,2448.792,658.883
BC00226=1984.483,2448.792,658.883
BC00227=1984.483,2448.792,658.883
BC00228=1984.483,2448.792,658.883
BC00229=1984.483,2448.792,658.883
BC00230=1984.483,2448.792,658.883
BC00231=1984.483,2448.792,658.883
BC00232=1984.483,2448.792,658.883
BC00233=1984.483,2448.792,658.883
BC00234=1984.483,2448.792,658.883
BC00235=1984.483,2448.792,658.883
BC00236=1984.483,2448.792,658.883
BC00237=1984.483,2448.792,658.883
BC00238=1984.483,2448.792,658.883
BC00239=1984.483,2448.792,658.883
BC00240=1984.483,2448.792,658.883
BC00241=1984.483,2020.544,658.883
BC00242=1984.483,2020.544,658.883
BC00243=1984.483,2020.544,658.883
BC00244=1984.483,2020.544,658.883
BC00245=1984.483,2020.544,658.883
BC00246=1984.483,2020.544,658.883
BC00247=1984.483,2020.544,658.883
BC00248=1984.470,2020.544,658.879
BC00249=1984.470,2020.544,658.879
BC00250=1984.470,2020.544,658.879
BC00251=1984.470,2020.544,658.879
BC00252=1984.470,2020.544,658.879
BC00253=1984.470,2020.544,658.879
BC00254=1984.470,2020.544,658.879
BC00255=1984.470,2020.544,658.879
BC00256=1984.470,2020.544,658.879
BC00257=1984.470,2020.544,658.879
BC00258=1984.470,2020.544,658.879
BC00259=1984.470,2020.538,658.877
BC00260=1391.860,3285.602,1013.728
BC00261=874.011,3770.839,1827.894
BC00262=779.962,3777.824,1999.134
BC00263=536.351,3774.159,1979.823
BC00264=1536.650,3350.624,1880.104
BC00265=2471.115,2623.215,1708.837
BC00266=2471.115,644.771,1708.837
BC00267=2471.115,644.771,371.374
BC00268=2499.895,888.831,371.374
BC00269=2499.895,888.831,371.366
BC00270=2499.895,888.831,371.366
BC00271=2499.895,888.831,371.366
BC00272=2499.895,888.831,371.366
BC00273=2499.895,888.831,371.366
BC00274=2499.895,888.831,371.366
BC00275=2499.895,888.831,371.366
BC00276=2499.895,888.825,371.363
BC00277=2499.895,888.825,371.363
BC00278=2499.895,888.825,371.363
BC00279=2499.895,888.825,371.363
BC00280=2499.895,888.825,371.363
BC00281=2499.895,888.825,371.363
BC00282=2499.895,888.825,371.363
BC00283=2499.895,888.825,371.363
BC00284=2499.895,888.825,371.363
BC00285=2499.895,888.825,371.363
BC00286=2499.895,888.825,371.363
BC00287=2499.895,648.814,371.363
BC00288=2499.895,648.814,371.363
BC00289=2499.895,648.814,371.363
BC00290=2499.895,648.814,371.363
BC00291=2499.895,648.814,371.363
BC00292=2499.895,648.814,371.363
BC00293=2499.895,648.814,371.363
BC00294=2499.895,648.814,371.363
BC00295=2499.895,648.814,371.363
BC00296=2499.895,648.814,371.363
BC00297=2499.895,648.814,371.363
BC00298=2499.895,648.814,371.363
BC00299=2499.895,648.814,371.363
BC00300=2499.895,648.814,371.363
BC00301=2499.895,648.814,371.363
BC00302=2499.895,648.814,371.363
BC00303=2499.895,972.335,371.363
BC00304=2499.895,972.335,371.363
BC00305=2499.895,972.335,371.363
BC00306=2204.921,409.519,319.294
BC00307=2204.921,409.519,319.294
BC00308=2204.921,409.519,319.294
BC00309=2204.921,409.519,319.294
BC00310=2204.921,409.519,319.294
BC00311=2204.921,409.519,319.294
BC00312=2204.921,409.519,319.294
BC00313=2493.165,409.519,1451.480
BC00314=2493.165,3204.728,1451.480
BC00315=430.297,4179.635,1999.619
///POSTYPE PULSE
///PULSE
EC00000=-811452,-554689
EC00001=-811450,-554689
EC00002=-811450,-554689
EC00003=-811450,-554689
EC00004=-811450,-554689
EC00005=-811450,-554689
EC00006=-811450,-554689
EC00007=-811450,-554689
EC00008=-811450,-554689
EC00009=-811450,-554689
EC00010=-811450,-554689
EC00011=-811450,-554689
EC00012=-811450,-554689
EC00013=-811450,-554689
EC00014=-811450,-554689
EC00015=-811450,-554689
EC00016=-811450,-554689
EC00017=-811450,-554689
EC00018=-811450,-554689
EC00019=-811450,-554689
EC00020=-811450,-554689
EC00021=-811450,-554689
EC00022=-811450,-554689
EC00023=-811450,-554689
EC00024=-811450,-554689
EC00025=-811450,-554689
EC00026=-811450,-554689
EC00027=-811450,-554689
EC00028=-811450,-554689
EC00029=-811450,-554689
EC00030=-811450,-554689
EC00031=-811450,-554689
EC00032=-811450,-554689
EC00033=-811450,-554689
EC00034=-811450,-554689
EC00035=-811450,-554689
EC00036=-811450,-554689
EC00037=-811450,-554689
EC00038=-811450,-554689
EC00039=-811450,-554689
EC00040=-811450,-554689
EC00041=-811450,-554689
EC00042=-811450,-554689
EC00043=-811450,-554689
EC00044=-811450,-554689
EC00045=-811450,-554689
EC00046=-811450,-554689
EC00047=-811450,-554689
EC00048=-811450,-554689
EC00049=-811450,-554689
EC00050=-811450,-554689
EC00051=-811450,-554689
EC00052=-811450,-554689
EC00053=-811450,-554689
EC00054=-811452,-554689
EC00055=-811452,-554689
EC00056=-811452,-554689
EC00057=-811451,-554689
EC00058=-811451,-554689
EC00059=-811451,-554689
EC00060=-811451,-554689
EC00061=-811451,-554689
EC00062=-811451,-554689
EC00063=-811451,-554689
EC00064=-811451,-554689
EC00065=-811451,-554689
EC00066=-811451,-554689
EC00067=-811451,-554689
EC00068=-811451,-554689
EC00069=-811451,-554689
EC00070=-811451,-554689
EC00071=-811451,-554689
EC00072=-811451,-554689
EC00073=-811451,-554689
EC00074=-811451,-554689
EC00075=-811451,-554689
EC00076=-811451,-554689
EC00077=-811451,-554689
EC00078=-811451,-554689
EC00079=-811451,-554689
EC00080=-811451,-554689
EC00081=-811451,-554689
EC00082=-811449,-554688
EC00083=-811451,-554689
EC00084=-811451,-554689
EC00085=-811451,-554689
EC00086=-811451,-554689
EC00087=-811451,-554689
EC00088=-811451,-554689
EC00089=-811451,-554689
EC00090=-811451,-554689
EC00091=-811451,-554689
EC00092=-811451,-554689
EC00093=-811451,-554689
EC00094=-811451,-554689
EC00095=-811451,-554689
EC00096=-811451,-554689
EC00097=-811451,-554689
EC00098=-811451,-554689
EC00099=-811451,-554689
EC00100=-811451,-554689
EC00101=-811451,-554689
EC00102=-363208,-550746
EC00103=-363208,-550746
EC00104=-363208,-550746
EC00105=-363208,-550746
EC00106=-363208,-550746
EC00107=-363208,-550746
EC00108=-363208,-550746
EC00109=-363208,-550746
EC00110=-363208,-550746
EC00111=-363208,-550746
EC00112=-363208,-550746
EC00113=-363208,-550746
EC00114=-363208,-550746
EC00115=-363208,-550746
EC00116=-363208,-550746
EC00117=-363208,-550746
EC00118=-363208,-550746
EC00119=-363208,-550746
EC00120=-363208,-550746
EC00121=-363208,-550746
EC00122=-363208,-550746
EC00123=-363208,-550746
EC00124=-363208,-550746
EC00125=-363208,-550746
EC00126=-363208,-550746
EC00127=-363208,-550746
EC00128=-363208,-550746
EC00129=-363208,-550746
EC00130=-363208,-550746
EC00131=-363208,-550746
EC00132=-363208,-550746
EC00133=-363208,-550746
EC00134=-363208,-550746
EC00135=-363208,-550746
EC00136=-363208,-550746
EC00137=-363208,-550746
EC00138=-363208,-550746
EC00139=-363208,-550746
EC00140=-363208,-550746
EC00141=-363208,-550746
EC00142=-363208,-550746
EC00143=-363208,-550746
EC00144=-363208,-550746
EC00145=-363208,-550746
EC00146=-363207,-550746
EC00147=-363207,-550746
EC00148=-363207,-550746
EC00149=-363207,-550746
EC00150=-363207,-550746
EC00151=-363207,-550746
EC00152=-363206,-550746
EC00153=-363206,-550746
EC00154=-363206,-550746
EC00155=-363206,-550746
EC00156=-363206,-550746
EC00157=-363206,-550746
EC00158=-363206,-550746
EC00159=-363206,-550746
EC00160=-363206,-550746
EC00161=-363206,-550746
EC00162=-363206,-550746
EC00163=-363206,-550746
EC00164=-363206,-550746
EC00165=-363206,-550746
EC00166=-363206,-550746
EC00167=-363206,-550746
EC00168=-363206,-550746
EC00169=-363206,-550746
EC00170=-363206,-550746
EC00171=-363206,-550746
EC00172=-363206,-550746
EC00173=-363206,-550746
EC00174=-363206,-550746
EC00175=-363206,-550746
EC00176=-363206,-550746
EC00177=-363206,-550746
EC00178=-363206,-550746
EC00179=-363206,-550746
EC00180=0,0
EC00181=-802750,0
EC00182=-802750,0
EC00183=-802750,0
EC00184=-802750,0
EC00185=-802750,0
EC00186=-802750,0
EC00187=-802750,0
EC00188=-802750,0
EC00189=-802750,0
EC00190=-802750,0
EC00191=-802750,0
EC00192=-802750,0
EC00193=-802750,0
EC00194=-802750,0
EC00195=-802750,0
EC00196=-802750,0
EC00197=-802750,0
EC00198=-802750,0
EC00199=-802750,0
EC00200=-802750,0
EC00201=-802750,0
EC00202=-802750,0
EC00203=-802750,0
EC00204=-802750,0
EC00205=-802750,0
EC00206=-802749,0
EC00207=-802749,0
EC00208=-802749,0
EC00209=-802749,0
EC00210=-802749,0
EC00211=-802749,0
EC00212=-802749,0
EC00213=-802749,0
EC00214=-802749,0
EC00215=-802749,0
EC00216=-802749,0
EC00217=-802748,0
EC00218=-802748,0
EC00219=793507,0
EC00220=793506,-1
EC00221=793506,-1
EC00222=793506,-1
EC00223=793506,-1
EC00224=793506,-1
EC00225=793506,-1
EC00226=793506,-1
EC00227=793505,-1
EC00228=793505,-1
EC00229=793505,-1
EC00230=793505,-1
EC00231=793505,-1
EC00232=793504,-1
EC00233=793504,-1
EC00234=793504,-1
EC00235=793504,-1
EC00236=793504,-1
EC00237=793504,-1
EC00238=793504,-1
EC00239=793504,-1
EC00240=793504,-1
EC00241=793504,-1
EC00242=793504,-1
EC00243=793504,-1
EC00244=793504,-1
EC00245=793504,-1
EC00246=793504,-1
EC00247=793504,-1
EC00248=793504,-1
EC00249=793504,-1
EC00250=793504,-1
EC00251=793504,-1
EC00252=793504,-1
EC00253=793504,-1
EC00254=793504,-1
EC00255=793504,-1
EC00256=793504,-1
EC00257=793504,-1
EC00258=793504,-1
EC00259=793504,-1
EC00260=793504,-1
EC00261=793504,-1
EC00262=793504,-1
EC00263=0,-1
///POSTYPE BASE
///RECTAN
///RCONF 0,0,0,0,1,0,0,0,0,0,0,0,0,0,0,0,0,0,0,0,0,0,0,0
P00006=2.006,1.622,-0.565,0.0000,0.0000,0.0000
P00021=0.073,2.058,-0.109,0.0000,0.0000,0.0000
P00022=2.006,1.622,-0.565,0.0000,0.0000,0.0000
///RCONF 0,0,0,0,0,0,0,0,0,0,0,0,0,0,0,0,0,0,0,0,0,0,0,0
P00023=-2.957,-4.083,2.762,0.0000,0.0000,0.0000
P00024=-1.466,-0.226,-0.419,0.0000,0.0000,0.0000
P00025=3.643,0.007,-2.585,0.0000,0.0000,0.0000
P00026=2.644,0.055,-2.583,0.0000,0.0000,0.0000
P00027=2.278,0.099,-4.210,0.0000,0.0000,0.0000
P00028=-1.778,-0.182,-2.050,0.0000,0.0000,0.0000
P00029=1.749,4.006,-0.261,0.0000,0.0000,0.0000
P00030=-0.014,-0.768,0.131,0.0000,0.0000,0.0000
P00031=-0.170,0.039,-0.647,0.0000,0.0000,0.0000
///RCONF 0,0,0,0,1,0,0,0,0,0,0,0,0,0,0,0,0,0,0,0,0,0,0,0
P00034=-8.151,9.743,-4.393,0.0000,0.0000,0.0000
///RCONF 0,0,0,0,0,0,0,0,0,0,0,0,0,0,0,0,0,0,0,0,0,0,0,0
P00035=0.390,-0.027,1.040,0.0000,0.0000,0.0000
P00036=-2.434,0.084,0.197,0.0000,0.0000,0.0000
P00037=-1.075,5.090,-3.949,0.0000,0.0000,0.0000
//INST
///DATE 2023/12/21 13:23
///ATTR SC,RW,RJ
////FRAME ROBOT
///GROUP1 RB1,BS1
///GROUP2 ST1
NOP
SFTOF
MOVJ C00000 BC00000 VJ=100.00  +MOVJ EC00000 VJ=100.00
'SZUKANIE
SFTOF
MOVL C00001 BC00001 V=83.3  +MOVJ EC00001 VJ=15.00
MOVL C00002 BC00002 V=83.3  +MOVJ EC00002 VJ=15.00
REFP 3 RB1 C00003 BC00003
CALL JOB:SEARCH-R1
SET P025 P006
SFTON P025
MOVL C00004 BC00004 V=83.3  +MOVJ EC00003 VJ=15.00
REFP 3 RB1 C00005 BC00005
CALL JOB:SEARCH-R1
SET P025 P006
MOVL C00006 BC00006 V=83.3  +MOVJ EC00004 VJ=15.00
SFTOF
MOVL C00007 BC00007 V=83.3  +MOVJ EC00005 VJ=15.00
MOVL C00008 BC00008 V=83.3  +MOVJ EC00006 VJ=15.00
REFP 3 RB1 C00009 BC00009
CALL JOB:SEARCH-R1
SET P026 P006
SFTON P026
MOVL C00010 BC00010 V=83.3  +MOVJ EC00007 VJ=15.00
REFP 3 RB1 C00011 BC00011
CALL JOB:SEARCH-R1
SET P026 P006
MOVL C00012 BC00012 V=83.3  +MOVJ EC00008 VJ=15.00
SFTOF
MOVL C00013 BC00013 V=83.3  +MOVJ EC00009 VJ=15.00
MOVL C00014 BC00014 V=83.3  +MOVJ EC00010 VJ=15.00
MOVL C00015 BC00015 V=83.3  +MOVJ EC00011 VJ=15.00
REFP 3 RB1 C00016 BC00016
CALL JOB:SEARCH-R1
SET P027 P006
SFTON P027
MOVL C00017 BC00017 V=83.3  +MOVJ EC00012 VJ=15.00
REFP 3 RB1 C00018 BC00018
CALL JOB:SEARCH-R1
SET P027 P006
MOVL C00019 BC00019 V=83.3  +MOVJ EC00013 VJ=15.00
SFTOF
MOVL C00020 BC00020 V=83.3  +MOVJ EC00014 VJ=15.00
MOVL C00021 BC00021 V=83.3  +MOVJ EC00015 VJ=15.00
REFP 3 RB1 C00022 BC00022
CALL JOB:SEARCH-R1
SET P028 P006
SFTON P028
MOVL C00023 BC00023 V=83.3  +MOVJ EC00016 VJ=15.00
REFP 3 RB1 C00024 BC00024
CALL JOB:SEARCH-R1
SET P028 P006
MOVL C00025 BC00025 V=83.3  +MOVJ EC00017 VJ=15.00
SFTOF
MOVL C00026 BC00026 V=83.3  +MOVJ EC00018 VJ=15.00
MOVL C00027 BC00027 V=83.3  +MOVJ EC00019 VJ=15.00
MOVL C00028 BC00028 V=83.3  +MOVJ EC00020 VJ=15.00
REFP 3 RB1 C00029 BC00029
CALL JOB:SEARCH-R1
SET P029 P006
SFTON P029
MOVL C00030 BC00030 V=83.3  +MOVJ EC00021 VJ=15.00
REFP 3 RB1 C00031 BC00031
CALL JOB:SEARCH-R1
SET P029 P006
MOVL C00032 BC00032 V=83.3  +MOVJ EC00022 VJ=15.00
SFTOF
MOVL C00033 BC00033 V=83.3  +MOVJ EC00023 VJ=15.00
MOVL C00034 BC00034 V=83.3  +MOVJ EC00024 VJ=15.00
MOVL C00035 BC00035 V=83.3  +MOVJ EC00025 VJ=15.00
REFP 3 RB1 C00036 BC00036
CALL JOB:SEARCH-R1
SET P030 P006
SFTON P030
MOVL C00037 BC00037 V=83.3  +MOVJ EC00026 VJ=15.00
REFP 3 RB1 C00038 BC00038
CALL JOB:SEARCH-R1
SET P030 P006
MOVL C00039 BC00039 V=83.3  +MOVJ EC00027 VJ=15.00
SFTOF
MOVL C00040 BC00040 V=83.3  +MOVJ EC00028 VJ=15.00
MOVL C00041 BC00041 V=83.3  +MOVJ EC00029 VJ=15.00
REFP 3 RB1 C00042 BC00042
CALL JOB:SEARCH-R1
SET P031 P006
SFTON P031
MOVL C00043 BC00043 V=83.3  +MOVJ EC00030 VJ=15.00
REFP 3 RB1 C00044 BC00044
CALL JOB:SEARCH-R1
SET P031 P006
MOVL C00045 BC00045 V=83.3  +MOVJ EC00031 VJ=15.00
SFTOF
MOVL C00046 BC00046 V=250.0  +MOVJ EC00032 VJ=15.00
MOVL C00047 BC00047 V=83.3  +MOVJ EC00033 VJ=15.00
REFP 3 RB1 C00048 BC00048
CALL JOB:SEARCH-R1
SET P036 P006
SFTON P036
MOVL C00049 BC00049 V=83.3  +MOVJ EC00034 VJ=15.00
REFP 3 RB1 C00050 BC00050
CALL JOB:SEARCH-R1
SET P036 P006
MOVL C00051 BC00051 V=83.3  +MOVJ EC00035 VJ=15.00
SFTOF
MOVL C00052 BC00052 V=250.0  +MOVJ EC00036 VJ=15.00
MOVJ C00053 BC00053 VJ=100.00  +MOVJ EC00037 VJ=15.00
MOVJ C00054 BC00054 VJ=100.00  +MOVJ EC00038 VJ=100.00
MOVJ C00055 BC00055 VJ=100.00  +MOVJ EC00039 VJ=100.00
MOVL C00056 BC00056 V=83.3  +MOVJ EC00040 VJ=15.00
REFP 3 RB1 C00057 BC00057
CALL JOB:SEARCH-R1
SET P037 P006
SFTON P037
MOVL C00058 BC00058 V=83.3  +MOVJ EC00041 VJ=15.00
REFP 3 RB1 C00059 BC00059
CALL JOB:SEARCH-R1
SET P037 P006
MOVL C00060 BC00060 V=83.3  +MOVJ EC00042 VJ=15.00
SFTOF
MOVL C00061 BC00061 V=166.7  +MOVJ EC00043 VJ=15.00
SFTON P037
MACRO1 MJ#(0) ARGF7
MOVL C00062 BC00062 V=83.3  +MOVJ EC00044 VJ=100.00
ARCON
MOVL C00063 BC00063 V=10.0  +MOVJ EC00045 VJ=100.00
MOVL C00064 BC00064 V=10.0  +MOVJ EC00046 VJ=100.00
MOVL C00065 BC00065 V=10.0  +MOVJ EC00047 VJ=100.00
MOVL C00066 BC00066 V=10.0  +MOVJ EC00048 VJ=100.00
MOVL C00067 BC00067 V=10.0  +MOVJ EC00049 VJ=100.00
MOVL C00068 BC00068 V=10.0  +MOVJ EC00050 VJ=100.00
SFTOF
MOVL C00069 BC00069 V=10.0  +MOVJ EC00051 VJ=100.00
MACRO1 MJ#(0) ARGF7
MOVL C00070 BC00070 V=10.0  +MOVJ EC00052 VJ=100.00
MOVL C00071 BC00071 V=10.0  +MOVJ EC00053 VJ=100.00
MOVL C00072 BC00072 V=10.0  +MOVJ EC00054 VJ=100.00
MOVL C00073 BC00073 V=10.0  +MOVJ EC00055 VJ=20.00
ARCOF
MOVJ C00074 BC00074 VJ=20.00  +MOVJ EC00056 VJ=20.00
SFTOF
MOVJ C00075 BC00075 VJ=100.00  +MOVJ EC00057 VJ=20.00
MOVJ C00076 BC00076 VJ=100.00  +MOVJ EC00058 VJ=20.00
SFTON P036
MOVJ C00077 BC00077 VJ=20.00  +MOVJ EC00059 VJ=100.00
ARCON
MOVL C00078 BC00078 V=10.0  +MOVJ EC00060 VJ=20.00
MOVL C00079 BC00079 V=10.0  +MOVJ EC00061 VJ=20.00
MOVL C00080 BC00080 V=10.0  +MOVJ EC00062 VJ=20.00
MOVL C00081 BC00081 V=10.0  +MOVJ EC00063 VJ=20.00
MOVL C00082 BC00082 V=10.0  +MOVJ EC00064 VJ=20.00
MOVL C00083 BC00083 V=10.0  +MOVJ EC00065 VJ=20.00
MOVL C00084 BC00084 V=10.0  +MOVJ EC00066 VJ=20.00
SFTOF
MOVL C00085 BC00085 V=10.0  +MOVJ EC00067 VJ=20.00
MOVL C00086 BC00086 V=10.0  +MOVJ EC00068 VJ=20.00
MOVL C00087 BC00087 V=10.0  +MOVJ EC00069 VJ=50.00
MOVL C00088 BC00088 V=10.0  +MOVJ EC00070 VJ=15.00
ARCOF
MOVJ C00089 BC00089 VJ=15.00  +MOVJ EC00071 VJ=15.00
SFTOF
MOVJ C00090 BC00090 VJ=100.00  +MOVJ EC00072 VJ=20.00
SFTON P028
MOVJ C00091 BC00091 VJ=20.00  +MOVJ EC00073 VJ=20.00
ARCON
MOVL C00092 BC00092 V=8.3  +MOVJ EC00074 VJ=20.00
SFTON P027
MOVL C00093 BC00093 V=10.0  +MOVJ EC00075 VJ=20.00
MOVL C00094 BC00094 V=10.0  +MOVJ EC00076 VJ=20.00
MOVL C00095 BC00095 V=10.0  +MOVJ EC00077 VJ=100.00
MOVL C00096 BC00096 V=10.0  +MOVJ EC00078 VJ=20.00
SFTON P026
MOVL C00097 BC00097 V=10.0  +MOVJ EC00079 VJ=20.00
MOVL C00098 BC00098 V=10.0  +MOVJ EC00080 VJ=20.00
MOVL C00099 BC00099 V=10.8  +MOVJ EC00081 VJ=20.00
MOVL C00100 BC00100 V=10.8  +MOVJ EC00082 VJ=20.00
SFTON P025
MOVL C00101 BC00101 V=10.8  +MOVJ EC00083 VJ=20.00
MOVL C00102 BC00102 V=10.8  +MOVJ EC00084 VJ=20.00
ARCOF
MOVJ C00103 BC00103 VJ=20.00  +MOVJ EC00085 VJ=20.00
SFTOF
MOVJ C00104 BC00104 VJ=100.00  +MOVJ EC00086 VJ=20.00
MOVJ C00105 BC00105 VJ=100.00  +MOVJ EC00087 VJ=20.00
SFTON P028
MOVJ C00106 BC00106 VJ=20.00  +MOVJ EC00088 VJ=20.00
ARCON
MOVL C00107 BC00107 V=10.0  +MOVJ EC00089 VJ=20.00
SFTON P029
MOVL C00108 BC00108 V=10.0  +MOVJ EC00090 VJ=20.00
MOVL C00109 BC00109 V=10.0  +MOVJ EC00091 VJ=20.00
MOVL C00110 BC00110 V=10.0  +MOVJ EC00092 VJ=20.00
MOVL C00111 BC00111 V=10.0  +MOVJ EC00093 VJ=20.00
SFTON P030
MOVL C00112 BC00112 V=10.0  +MOVJ EC00094 VJ=20.00
MOVL C00113 BC00113 V=10.0  +MOVJ EC00095 VJ=20.00
MOVL C00114 BC00114 V=10.0  +MOVJ EC00096 VJ=20.00
MOVL C00115 BC00115 V=10.0  +MOVJ EC00097 VJ=20.00
SFTON P031
MOVL C00116 BC00116 V=10.0  +MOVJ EC00098 VJ=20.00
MOVL C00117 BC00117 V=10.0  +MOVJ EC00099 VJ=20.00
ARCOF
MOVJ C00118 BC00118 VJ=20.00  +MOVJ EC00100 VJ=20.00
SFTOF
MOVJ C00119 BC00119 VJ=100.00  +MOVJ EC00101 VJ=100.00
MOVJ C00120 BC00120 VJ=100.00  +MOVJ EC00102 VJ=100.00
CALL JOB:CLEAN-R1_LONG
MOVJ C00121 BC00121 VJ=100.00  +MOVJ EC00103 VJ=100.00
MOVJ C00122 BC00122 VJ=100.00  +MOVJ EC00104 VJ=100.00
'SZUKANIE DRUGA STRONA
MOVJ C00123 BC00123 VJ=30.00  +MOVJ EC00105 VJ=15.00
SFTOF
MOVL C00124 BC00124 V=83.3  +MOVJ EC00106 VJ=15.00
REFP 3 RB1 C00125 BC00125
CALL JOB:SEARCH-R1
SET P035 P006
SFTON P035
MOVL C00126 BC00126 V=83.3  +MOVJ EC00107 VJ=15.00
REFP 3 RB1 C00127 BC00127
CALL JOB:SEARCH-R1
SET P035 P006
MOVL C00128 BC00128 V=83.3  +MOVJ EC00108 VJ=15.00
SFTOF
MOVJ C00129 BC00129 VJ=50.00  +MOVJ EC00109 VJ=50.00
MOVJ C00130 BC00130 VJ=15.00  +MOVJ EC00110 VJ=15.00
MOVL C00131 BC00131 V=83.3  +MOVJ EC00111 VJ=15.00
REFP 3 RB1 C00132 BC00132
CALL JOB:SEARCH-R1
SET P025 P006
SFTON P025
MOVL C00133 BC00133 V=83.3  +MOVJ EC00112 VJ=15.00
REFP 3 RB1 C00134 BC00134
CALL JOB:SEARCH-R1
SET P025 P006
MOVL C00135 BC00135 V=83.3  +MOVJ EC00113 VJ=15.00
SFTOF
MOVL C00136 BC00136 V=83.3  +MOVJ EC00114 VJ=15.00
MOVL C00137 BC00137 V=83.3  +MOVJ EC00115 VJ=15.00
REFP 3 RB1 C00138 BC00138
CALL JOB:SEARCH-R1
SET P026 P006
SFTON P026
MOVL C00139 BC00139 V=83.3  +MOVJ EC00116 VJ=15.00
REFP 3 RB1 C00140 BC00140
CALL JOB:SEARCH-R1
SET P026 P006
MOVL C00141 BC00141 V=83.3  +MOVJ EC00117 VJ=15.00
SFTOF
MOVL C00142 BC00142 V=83.3  +MOVJ EC00118 VJ=15.00
MOVL C00143 BC00143 V=83.3  +MOVJ EC00119 VJ=15.00
REFP 3 RB1 C00144 BC00144
CALL JOB:SEARCH-R1
SET P027 P006
SFTON P027
MOVL C00145 BC00145 V=83.3  +MOVJ EC00120 VJ=15.00
REFP 3 RB1 C00146 BC00146
CALL JOB:SEARCH-R1
SET P027 P006
MOVL C00147 BC00147 V=83.3  +MOVJ EC00121 VJ=15.00
SFTOF
MOVL C00148 BC00148 V=83.3  +MOVJ EC00122 VJ=15.00
MOVL C00149 BC00149 V=83.3  +MOVJ EC00123 VJ=15.00
REFP 3 RB1 C00150 BC00150
CALL JOB:SEARCH-R1
SET P028 P006
SFTON P028
MOVL C00151 BC00151 V=83.3  +MOVJ EC00124 VJ=15.00
REFP 3 RB1 C00152 BC00152
CALL JOB:SEARCH-R1
SET P028 P006
MOVL C00153 BC00153 V=83.3  +MOVJ EC00125 VJ=15.00
SFTOF
MOVL C00154 BC00154 V=83.3  +MOVJ EC00126 VJ=15.00
MOVL C00155 BC00155 V=83.3  +MOVJ EC00127 VJ=15.00
REFP 3 RB1 C00156 BC00156
CALL JOB:SEARCH-R1
SET P029 P006
SFTON P029
MOVL C00157 BC00157 V=83.3  +MOVJ EC00128 VJ=15.00
REFP 3 RB1 C00158 BC00158
CALL JOB:SEARCH-R1
SET P029 P006
MOVL C00159 BC00159 V=83.3  +MOVJ EC00129 VJ=15.00
SFTOF
MOVJ C00160 BC00160 VJ=15.00  +MOVJ EC00130 VJ=15.00
MOVJ C00161 BC00161 VJ=15.00  +MOVJ EC00131 VJ=15.00
SFTOF
MOVJ C00162 BC00162 VJ=15.00  +MOVJ EC00132 VJ=15.00
MOVL C00163 BC00163 V=83.3  +MOVJ EC00133 VJ=15.00
REFP 3 RB1 C00164 BC00164
CALL JOB:SEARCH-R1
SET P034 P006
SFTON P034
MOVL C00165 BC00165 V=83.3  +MOVJ EC00134 VJ=15.00
REFP 3 RB1 C00166 BC00166
CALL JOB:SEARCH-R1
SET P034 P006
MOVL C00167 BC00167 V=83.3  +MOVJ EC00135 VJ=15.00
MOVJ C00168 BC00168 VJ=15.00  +MOVJ EC00136 VJ=15.00
'KONIEC SZUKANIE DRUGA STRONA
'SPAWANIE DRUGA STRONA
MOVJ C00169 BC00169 VJ=15.00  +MOVJ EC00137 VJ=15.00
MACRO1 MJ#(0) ARGF7
SFTOF
SFTON P034
MOVJ C00170 BC00170 VJ=15.00  +MOVJ EC00138 VJ=15.00
ARCON
MOVL C00171 BC00171 V=10.0  +MOVJ EC00139 VJ=15.00
MOVL C00172 BC00172 V=10.0  +MOVJ EC00140 VJ=15.00
SFTOF
ARCOF
MOVJ C00173 BC00173 VJ=15.00  +MOVJ EC00141 VJ=15.00
MOVJ C00174 BC00174 VJ=50.00  +MOVJ EC00142 VJ=15.00
MOVJ C00175 BC00175 VJ=50.00  +MOVJ EC00143 VJ=50.00
MOVJ C00176 BC00176 VJ=50.00  +MOVJ EC00144 VJ=50.00
MOVJ C00177 BC00177 VJ=50.00  +MOVJ EC00145 VJ=50.00
SFTON P035
MOVL C00178 BC00178 V=83.3  +MOVJ EC00146 VJ=50.00
ARCON
MOVL C00179 BC00179 V=10.0  +MOVJ EC00147 VJ=50.00
MOVL C00180 BC00180 V=10.0  +MOVJ EC00148 VJ=50.00
ARCOF
SFTOF
MOVJ C00181 BC00181 VJ=20.00  +MOVJ EC00149 VJ=50.00
MOVJ C00182 BC00182 VJ=50.00  +MOVJ EC00150 VJ=20.00
SFTON P027
MOVJ C00183 BC00183 VJ=15.00  +MOVJ EC00151 VJ=50.00
ARCON
MOVL C00184 BC00184 V=10.0  +MOVJ EC00152 VJ=15.00
MOVL C00185 BC00185 V=10.0  +MOVJ EC00153 VJ=15.00
MOVL C00186 BC00186 V=10.0  +MOVJ EC00154 VJ=15.00
MOVL C00187 BC00187 V=10.0  +MOVJ EC00155 VJ=15.00
SFTON P028
MOVL C00188 BC00188 V=10.0  +MOVJ EC00156 VJ=15.00
MOVL C00189 BC00189 V=10.0  +MOVJ EC00157 VJ=15.00
MOVL C00190 BC00190 V=10.0  +MOVJ EC00158 VJ=15.00
MOVL C00191 BC00191 V=10.0  +MOVJ EC00159 VJ=15.00
SFTON P029
MOVL C00192 BC00192 V=10.0  +MOVJ EC00160 VJ=15.00
MOVL C00193 BC00193 V=10.0  +MOVJ EC00161 VJ=15.00
ARCOF
MOVJ C00194 BC00194 VJ=15.00  +MOVJ EC00162 VJ=15.00
MOVJ C00195 BC00195 VJ=15.00  +MOVJ EC00163 VJ=15.00
SFTOF
MOVJ C00196 BC00196 VJ=15.00  +MOVJ EC00164 VJ=15.00
SFTON P027
MOVJ C00197 BC00197 VJ=15.00  +MOVJ EC00165 VJ=15.00
ARCON
MOVL C00198 BC00198 V=10.0  +MOVJ EC00166 VJ=15.00
MOVL C00199 BC00199 V=10.0  +MOVJ EC00167 VJ=15.00
MOVL C00200 BC00200 V=10.0  +MOVJ EC00168 VJ=15.00
MOVL C00201 BC00201 V=10.0  +MOVJ EC00169 VJ=15.00
SFTON P026
MOVL C00202 BC00202 V=10.0  +MOVJ EC00170 VJ=15.00
MOVL C00203 BC00203 V=10.0  +MOVJ EC00171 VJ=15.00
MOVL C00204 BC00204 V=10.0  +MOVJ EC00172 VJ=15.00
MOVL C00205 BC00205 V=10.0  +MOVJ EC00173 VJ=15.00
SFTON P025
MOVL C00206 BC00206 V=10.0  +MOVJ EC00174 VJ=15.00
MOVL C00207 BC00207 V=10.0  +MOVJ EC00175 VJ=15.00
MOVL C00208 BC00208 V=10.0  +MOVJ EC00176 VJ=15.00
ARCOF
MOVJ C00209 BC00209 VJ=15.00  +MOVJ EC00177 VJ=15.00
SFTOF
MOVJ C00210 BC00210 VJ=100.00  +MOVJ EC00178 VJ=15.00
MOVJ C00211 BC00211 VJ=100.00  +MOVJ EC00179 VJ=100.00
MOVJ C00212 BC00212 VJ=100.00  +MOVJ EC00180 VJ=100.00
MOVJ C00213 BC00213 VJ=100.00  +MOVJ EC00181 VJ=100.00
CALL JOB:CLEAN-R1_LONG
MOVJ C00214 BC00214 VJ=100.00  +MOVJ EC00182 VJ=100.00
MOVJ C00215 BC00215 VJ=100.00  +MOVJ EC00183 VJ=100.00
MOVJ C00216 BC00216 VJ=100.00  +MOVJ EC00184 VJ=100.00
MOVL C00217 BC00217 V=83.3  +MOVJ EC00185 VJ=15.00
REFP 3 RB1 C00218 BC00218
CALL JOB:SEARCH-R1
SET P021 P006
SFTON P021
MOVL C00219 BC00219 V=83.3  +MOVJ EC00186 VJ=15.00
REFP 3 RB1 C00220 BC00220
CALL JOB:SEARCH-R1
SET P021 P006
MOVL C00221 BC00221 V=83.3  +MOVJ EC00187 VJ=15.00
SFTOF
MOVL C00222 BC00222 V=166.7  +MOVJ EC00188 VJ=15.00
MOVL C00223 BC00223 V=83.3  +MOVJ EC00189 VJ=15.00
REFP 3 RB1 C00224 BC00224
CALL JOB:SEARCH-R1
SET P022 P006
SFTON P022
MOVL C00225 BC00225 V=83.3  +MOVJ EC00190 VJ=15.00
REFP 3 RB1 C00226 BC00226
CALL JOB:SEARCH-R1
SET P022 P006
MOVL C00227 BC00227 V=83.3  +MOVJ EC00191 VJ=15.00
SFTOF
MOVL C00228 BC00228 V=166.7  +MOVJ EC00192 VJ=15.00
MOVL C00229 BC00229 V=83.3  +MOVJ EC00193 VJ=15.00
REFP 3 RB1 C00230 BC00230
CALL JOB:SEARCH-R1
SET P023 P006
SFTON P023
MOVL C00231 BC00231 V=83.3  +MOVJ EC00194 VJ=15.00
REFP 3 RB1 C00232 BC00232
CALL JOB:SEARCH-R1
SET P023 P006
MOVL C00233 BC00233 V=83.3  +MOVJ EC00195 VJ=15.00
SFTOF
MOVL C00234 BC00234 V=166.7  +MOVJ EC00196 VJ=15.00
MOVL C00235 BC00235 V=83.3  +MOVJ EC00197 VJ=15.00
REFP 3 RB1 C00236 BC00236
CALL JOB:SEARCH-R1
SET P024 P006
SFTON P024
MOVL C00237 BC00237 V=83.3  +MOVJ EC00198 VJ=15.00
REFP 3 RB1 C00238 BC00238
CALL JOB:SEARCH-R1
SET P024 P006
MOVL C00239 BC00239 V=83.3  +MOVJ EC00199 VJ=15.00
SFTOF
MOVL C00240 BC00240 V=166.7  +MOVJ EC00200 VJ=15.00
MOVL C00241 BC00241 V=83.3  +MOVJ EC00201 VJ=15.00
REFP 3 RB1 C00242 BC00242
CALL JOB:SEARCH-R1
SET P025 P006
SFTON P025
MOVL C00243 BC00243 V=83.3  +MOVJ EC00202 VJ=15.00
REFP 3 RB1 C00244 BC00244
CALL JOB:SEARCH-R1
SET P025 P006
MOVL C00245 BC00245 V=83.3  +MOVJ EC00203 VJ=15.00
SFTOF
MOVJ C00246 BC00246 VJ=30.00  +MOVJ EC00204 VJ=100.00
MOVJ C00247 BC00247 VJ=30.00  +MOVJ EC00205 VJ=30.00
SFTON P023
MACRO1 MJ#(0) ARGF7
MOVL C00248 BC00248 V=83.3  +MOVJ EC00206 VJ=30.00
ARCON
SFTON P022
MOVL C00249 BC00249 V=10.8  +MOVJ EC00207 VJ=30.00
SFTON P021
MOVL C00250 BC00250 V=10.8  +MOVJ EC00208 VJ=30.00
MOVL C00251 BC00251 V=10.8  +MOVJ EC00209 VJ=30.00
ARCOF
SFTOF
MOVJ C00252 BC00252 VJ=30.00  +MOVJ EC00210 VJ=30.00
MOVJ C00253 BC00253 VJ=30.00  +MOVJ EC00211 VJ=30.00
SFTON P023
MOVL C00254 BC00254 V=83.3  +MOVJ EC00212 VJ=30.00
ARCON
SFTON P024
MOVL C00255 BC00255 V=10.8  +MOVJ EC00213 VJ=30.00
SFTON P025
MOVL C00256 BC00256 V=10.8  +MOVJ EC00214 VJ=30.00
MOVL C00257 BC00257 V=10.8  +MOVJ EC00215 VJ=30.00
MOVL C00258 BC00258 V=10.8  +MOVJ EC00216 VJ=30.00
ARCOF
SFTOF
MOVJ C00259 BC00259 VJ=30.00  +MOVJ EC00217 VJ=30.00
MOVJ C00260 BC00260 VJ=30.00  +MOVJ EC00218 VJ=30.00
MOVJ C00261 BC00261 VJ=100.00  +MOVJ EC00219 VJ=100.00
MOVJ C00262 BC00262 VJ=30.00  +MOVJ EC00220 VJ=30.00
CALL JOB:ONLYCUT-R1_LONG
MOVJ C00263 BC00263 VJ=30.00  +MOVJ EC00221 VJ=30.00
MOVJ C00264 BC00264 VJ=100.00  +MOVJ EC00222 VJ=100.00
MOVJ C00265 BC00265 VJ=30.00  +MOVJ EC00223 VJ=30.00
MOVJ C00266 BC00266 VJ=30.00  +MOVJ EC00224 VJ=30.00
MOVJ C00267 BC00267 VJ=30.00  +MOVJ EC00225 VJ=30.00
MOVJ C00268 BC00268 VJ=30.00  +MOVJ EC00226 VJ=30.00
MOVJ C00269 BC00269 VJ=100.00  +MOVJ EC00227 VJ=100.00
MOVL C00270 BC00270 V=83.3  +MOVJ EC00228 VJ=15.00
REFP 3 RB1 C00271 BC00271
CALL JOB:SEARCH-R1
SET P021 P006
SFTON P021
MOVL C00272 BC00272 V=83.3  +MOVJ EC00229 VJ=15.00
REFP 3 RB1 C00273 BC00273
CALL JOB:SEARCH-R1
SET P021 P006
MOVL C00274 BC00274 V=83.3  +MOVJ EC00230 VJ=15.00
SFTOF
MOVL C00275 BC00275 V=166.7  +MOVJ EC00231 VJ=15.00
MOVL C00276 BC00276 V=83.3  +MOVJ EC00232 VJ=15.00
REFP 3 RB1 C00277 BC00277
CALL JOB:SEARCH-R1
SET P022 P006
SFTON P022
MOVL C00278 BC00278 V=83.3  +MOVJ EC00233 VJ=15.00
REFP 3 RB1 C00279 BC00279
CALL JOB:SEARCH-R1
SET P022 P006
MOVL C00280 BC00280 V=83.3  +MOVJ EC00234 VJ=15.00
SFTOF
MOVL C00281 BC00281 V=166.7  +MOVJ EC00235 VJ=15.00
MOVL C00282 BC00282 V=83.3  +MOVJ EC00236 VJ=15.00
REFP 3 RB1 C00283 BC00283
CALL JOB:SEARCH-R1
SET P023 P006
SFTON P023
MOVL C00284 BC00284 V=83.3  +MOVJ EC00237 VJ=15.00
REFP 3 RB1 C00285 BC00285
CALL JOB:SEARCH-R1
SET P023 P006
MOVL C00286 BC00286 V=83.3  +MOVJ EC00238 VJ=15.00
SFTOF
MOVL C00287 BC00287 V=166.7  +MOVJ EC00239 VJ=15.00
MOVL C00288 BC00288 V=83.3  +MOVJ EC00240 VJ=15.00
REFP 3 RB1 C00289 BC00289
CALL JOB:SEARCH-R1
SET P024 P006
SFTON P024
MOVL C00290 BC00290 V=83.3  +MOVJ EC00241 VJ=15.00
REFP 3 RB1 C00291 BC00291
CALL JOB:SEARCH-R1
SET P024 P006
MOVL C00292 BC00292 V=83.3  +MOVJ EC00242 VJ=15.00
SFTOF
MOVL C00293 BC00293 V=166.7  +MOVJ EC00243 VJ=15.00
MOVL C00294 BC00294 V=83.3  +MOVJ EC00244 VJ=15.00
REFP 3 RB1 C00295 BC00295
CALL JOB:SEARCH-R1
SET P025 P006
SFTON P025
MOVL C00296 BC00296 V=83.3  +MOVJ EC00245 VJ=15.00
REFP 3 RB1 C00297 BC00297
CALL JOB:SEARCH-R1
SET P025 P006
MOVL C00298 BC00298 V=83.3  +MOVJ EC00246 VJ=15.00
SFTOF
MOVJ C00299 BC00299 VJ=30.00  +MOVJ EC00247 VJ=100.00
MOVJ C00300 BC00300 VJ=30.00  +MOVJ EC00248 VJ=30.00
SFTON P023
MOVL C00301 BC00301 V=83.3  +MOVJ EC00249 VJ=30.00
ARCON
SFTON P022
MOVL C00302 BC00302 V=10.8  +MOVJ EC00250 VJ=30.00
SFTON P021
MOVL C00303 BC00303 V=10.8  +MOVJ EC00251 VJ=30.00
MOVL C00304 BC00304 V=10.8  +MOVJ EC00252 VJ=30.00
ARCOF
SFTOF
MOVJ C00305 BC00305 VJ=30.00  +MOVJ EC00253 VJ=30.00
MOVJ C00306 BC00306 VJ=30.00  +MOVJ EC00254 VJ=30.00
SFTON P023
MOVL C00307 BC00307 V=83.3  +MOVJ EC00255 VJ=30.00
ARCON
SFTON P024
MOVL C00308 BC00308 V=10.8  +MOVJ EC00256 VJ=30.00
SFTON P025
MOVL C00309 BC00309 V=10.8  +MOVJ EC00257 VJ=30.00
MOVL C00310 BC00310 V=10.8  +MOVJ EC00258 VJ=30.00
MOVL C00311 BC00311 V=10.8  +MOVJ EC00259 VJ=30.00
ARCOF
SFTOF
MOVJ C00312 BC00312 VJ=50.00  +MOVJ EC00260 VJ=30.00
MOVJ C00313 BC00313 VJ=50.00  +MOVJ EC00261 VJ=30.00
MOVJ C00314 BC00314 VJ=50.00  +MOVJ EC00262 VJ=30.00
MOVJ C00315 BC00315 VJ=100.00  +MOVJ EC00263 VJ=30.00
END
